(* IEC 61131-3 sources: CodesysTest/export/SX.dev/Plc Logic/Application/DeviceController.pou/Communication States, 3 files *)

(* ---- Reset.m.st ---- *)
(*#-#-#-#-#-#-#-#-#-#---Declaration---#-#-#-#-#-#-#-#-#-#-#-#-#*)

(* Reset a device *)
METHOD PUBLIC Reset : DED.ERROR
VAR_INPUT
	itfDevice : DED.IDevice2;
END_VAR
(*#-#-#-#-#-#-#-#-#-#---Implementation---#-#-#-#-#-#-#-#-#-#-#-#-#*)

IF itfDevice <> 0 THEN

	(* with CheckSupportedCommunicationState() it is possible to check whether the requested state can be performed in general. *)
	IF itfDevice.CheckSupportedCommunicationState(DED.DEVICE_TRANSITION_STATE.RESET) THEN

		(* with CheckCurrentSupportedCommunicationState() it is possible to check whether the device can be reset right now. *)
		IF itfDevice.CheckCurrentSupportedCommunicationState(DED.DEVICE_TRANSITION_STATE.RESET) THEN
			(* reset the device*)
			itfDevice.SetCommunicationState(DED.DEVICE_TRANSITION_STATE.RESET);
		ELSE
			(* device is not ready to be reset. *)
			Reset := DED.ERROR.OPERATION_INVALID;
		END_IF
	ELSE
		(* device does not support "Reset" *)
		Reset := DED.ERROR.NOT_SUPPORTED;
	END_IF

END_IF

(* ---- Start.m.st ---- *)
(*#-#-#-#-#-#-#-#-#-#---Declaration---#-#-#-#-#-#-#-#-#-#-#-#-#*)

(* Start a device *)
METHOD PUBLIC Start : DED.ERROR
VAR_INPUT
	itfDevice : DED.IDevice2;
END_VAR
(*#-#-#-#-#-#-#-#-#-#---Implementation---#-#-#-#-#-#-#-#-#-#-#-#-#*)

IF itfDevice <> 0 THEN

	(* with CheckSupportedCommunicationState() it is possible to check whether the requested state can be performed in general. *)
	IF itfDevice.CheckSupportedCommunicationState(DED.DEVICE_TRANSITION_STATE.START) THEN

		(* with CheckCurrentSupportedCommunicationState() it is possible to check whether the device can be started right now. *)
		IF itfDevice.CheckCurrentSupportedCommunicationState(DED.DEVICE_TRANSITION_STATE.START) THEN
			(* start the device *)
			itfDevice.SetCommunicationState(DED.DEVICE_TRANSITION_STATE.START);
		ELSE
			(* device is not ready to start. *)
			Start := DED.ERROR.OPERATION_INVALID;
		END_IF
	ELSE
		(* device does not support "Start" *)
		Start := DED.ERROR.NOT_SUPPORTED;
	END_IF

END_IF

(* ---- Stop.m.st ---- *)
(*#-#-#-#-#-#-#-#-#-#---Declaration---#-#-#-#-#-#-#-#-#-#-#-#-#*)

(* Stop a device *)
METHOD PUBLIC Stop : DED.ERROR
VAR_INPUT
	itfDevice : DED.IDevice2;
END_VAR
(*#-#-#-#-#-#-#-#-#-#---Implementation---#-#-#-#-#-#-#-#-#-#-#-#-#*)

IF itfDevice <> 0 THEN

	(* with CheckSupportedCommunicationState() it is possible to check whether the requested state can be performed in general. *)
	IF itfDevice.CheckSupportedCommunicationState(DED.DEVICE_TRANSITION_STATE.STOP) THEN

		(* with CheckCurrentSupportedCommunicationState() it is possible to check whether the device can be stopped right now. *)
		IF itfDevice.CheckCurrentSupportedCommunicationState(DED.DEVICE_TRANSITION_STATE.STOP) THEN
			(* stop the device *)
			itfDevice.SetCommunicationState(DED.DEVICE_TRANSITION_STATE.STOP);
		ELSE
			(* device is not ready to be stopped. *)
			Stop := DED.ERROR.OPERATION_INVALID;
		END_IF
	ELSE
		(* device does not support "Stop" *)
		Stop := DED.ERROR.NOT_SUPPORTED;
	END_IF

END_IF
